  MoveL 7193 to (-68.89, 13.92, -254.44) mm, rotated rx 81.04 ry 30.21 rz 20.91 deg; joints [-4.482, -3.085, 63.14, 103.728, 105.898, 55.876, -153.967]
  MoveL 7194 to (-69.18, 14.22, -254.5) mm, rotated rx 81.04 ry 30.21 rz 20.91 deg; joints [-4.474, -3.068, 63.132, 103.732, 105.896, 55.866, -153.967]
  MoveL 7195 to (-69.51, 14.55, -254.53) mm, rotated rx 81.04 ry 30.21 rz 20.91 deg; joints [-4.464, -3.052, 63.128, 103.737, 105.894, 55.854, -153.967]
  MoveL 7196 to (-69.85, 14.88, -254.55) mm, rotated rx 81.04 ry 30.21 rz 20.91 deg; joints [-4.454, -3.036, 63.123, 103.743, 105.892, 55.84, -153.967]
  MoveL 7197 to (-70.15, 15.2, -254.6) mm, rotated rx 81.04 ry 30.21 rz 20.91 deg; joints [-4.445, -3.02, 63.118, 103.747, 105.89, 55.829, -153.967]
  MoveL 7198 to (-70.42, 15.5, -254.66) mm, rotated rx 81.04 ry 30.21 rz 20.91 deg; joints [-4.438, -3.004, 63.111, 103.751, 105.889, 55.819, -153.967]
  MoveL 7199 to (-70.7, 15.8, -254.71) mm, rotated rx 81.04 ry 30.21 rz 20.91 deg; joints [-4.43, -2.989, 63.105, 103.755, 105.887, 55.808, -153.967]
  MoveL 7200 to (-71.01, 16.11, -254.74) mm, rotated rx 81.04 ry 30.21 rz 20.91 deg; joints [-4.421, -2.973, 63.1, 103.759, 105.885, 55.796, -153.967]
  MoveL 7201 to (-71.4, 16.46, -254.74) mm, rotated rx 81.04 ry 30.21 rz 20.91 deg; joints [-4.409, -2.958, 63.098, 103.766, 105.882, 55.781, -153.967]
  MoveL 7202 to (-73.37, 18.61, -255.1) mm, rotated rx 81.04 ry 30.21 rz 20.91 deg; joints [-4.352, -2.846, 63.055, 103.794, 105.871, 55.705, -153.967]
  MoveL 7203 to (-74.08, 19.69, -255.54) mm, rotated rx 81.04 ry 30.21 rz 20.91 deg; joints [-4.336, -2.778, 63.012, 103.801, 105.869, 55.678, -153.967]
  MoveL 7204 to (-74.6, 20.77, -256.16) mm, rotated rx 81.04 ry 30.21 rz 20.91 deg; joints [-4.327, -2.701, 62.953, 103.803, 105.87, 55.658, -153.967]
  MoveL 7205 to (-75.09, 22.93, -257.95) mm, rotated rx 81.04 ry 30.21 rz 20.91 deg; joints [-4.333, -2.52, 62.791, 103.793, 105.877, 55.64, -153.967]
  MoveL 7206 to (-74.84, 25.11, -260.44) mm, rotated rx 81.04 ry 30.21 rz 20.91 deg; joints [-4.37, -2.305, 62.568, 103.764, 105.893, 55.652, -153.967]
  MoveL 7207 to (-74.04, 26.72, -262.93) mm, rotated rx 81.04 ry 30.21 rz 20.91 deg; joints [-4.424, -2.113, 62.345, 103.728, 105.912, 55.691, -153.967]
  MoveL 7208 to (-73.5, 27.09, -263.91) mm, rotated rx 81.04 ry 30.21 rz 20.91 deg; joints [-4.452, -2.047, 62.256, 103.711, 105.92, 55.717, -153.967]
  MoveL 7209 to (-72.87, 27.18, -264.71) mm, rotated rx 81.04 ry 30.21 rz 20.91 deg; joints [-4.481, -2.001, 62.182, 103.694, 105.927, 55.749, -153.967]
  MoveL 7210 to (-72.52, 27.12, -265.05) mm, rotated rx 81.04 ry 30.21 rz 20.91 deg; joints [-4.496, -1.986, 62.151, 103.687, 105.93, 55.767, -153.967]
  MoveL 7211 to (-72.14, 26.98, -265.34) mm, rotated rx 81.04 ry 30.21 rz 20.91 deg; joints [-4.51, -1.976, 62.123, 103.679, 105.933, 55.786, -153.967]
  MoveL 7212 to (-71.33, 26.5, -265.78) mm, rotated rx 81.04 ry 30.21 rz 20.91 deg; joints [-4.541, -1.97, 62.08, 103.664, 105.939, 55.828, -153.967]
  MoveL 7213 to (-70.42, 25.73, -266.05) mm, rotated rx 81.04 ry 30.21 rz 20.91 deg; joints [-4.572, -1.985, 62.052, 103.65, 105.944, 55.876, -153.967]
  MoveL 7214 to (-69.43, 24.68, -266.14) mm, rotated rx 81.04 ry 30.21 rz 20.91 deg; joints [-4.603, -2.02, 62.039, 103.637, 105.948, 55.928, -153.967]
  MoveL 7215 to (-67.7, 22.71, -266.14) mm, rotated rx 81.04 ry 30.21 rz 20.91 deg; joints [-4.656, -2.094, 62.03, 103.617, 105.954, 56.018, -153.967]
  MoveL 7216 to (-67.43, 22.36, -266.11) mm, rotated rx 81.04 ry 30.21 rz 20.91 deg; joints [-4.664, -2.109, 62.032, 103.614, 105.955, 56.032, -153.967]
  MoveL 7217 to (-67.18, 22.04, -266.06) mm, rotated rx 81.04 ry 30.21 rz 20.91 deg; joints [-4.671, -2.124, 62.035, 103.611, 105.956, 56.045, -153.967]
  MoveL 7218 to (-66.95, 21.73, -265.99) mm, rotated rx 81.04 ry 30.21 rz 20.91 deg; joints [-4.677, -2.14, 62.041, 103.609, 105.956, 56.056, -153.967]
  MoveL 7219 to (-66.69, 21.39, -265.94) mm, rotated rx 81.04 ry 30.21 rz 20.91 deg; joints [-4.685, -2.155, 62.044, 103.606, 105.957, 56.069, -153.967]
  MoveL 7220 to (-66.38, 21, -265.9) mm, rotated rx 81.04 ry 30.21 rz 20.91 deg; joints [-4.694, -2.172, 62.046, 103.602, 105.958, 56.085, -153.967]
  MoveL 7221 to (-66.06, 20.59, -265.84) mm, rotated rx 81.04 ry 30.21 rz 20.91 deg; joints [-4.703, -2.191, 62.05, 103.599, 105.959, 56.102, -153.967]
  MoveL 7222 to (-65.71, 20.17, -265.83) mm, rotated rx 81.04 ry 30.21 rz 20.91 deg; joints [-4.713, -2.208, 62.05, 103.595, 105.96, 56.12, -153.967]
  MoveL 7223 to (-65.28, 19.69, -265.84) mm, rotated rx 81.04 ry 30.21 rz 20.91 deg; joints [-4.727, -2.225, 62.046, 103.59, 105.961, 56.143, -153.967]
  MoveL 7224 to (-64.69, 19.05, -265.91) mm, rotated rx 81.04 ry 30.21 rz 20.91 deg; joints [-4.745, -2.244, 62.035, 103.583, 105.963, 56.176, -153.967]
  MoveL 7225 to (-64.35, 18.66, -265.91) mm, rotated rx 81.04 ry 30.21 rz 20.91 deg; joints [-4.756, -2.259, 62.033, 103.579, 105.965, 56.194, -153.967]
  MoveL 7226 to (-64.02, 18.28, -265.9) mm, rotated rx 81.04 ry 30.21 rz 20.91 deg; joints [-4.766, -2.273, 62.031, 103.575, 105.966, 56.211, -153.967]
  MoveL 7227 to (-63.72, 17.92, -265.88) mm, rotated rx 81.04 ry 30.21 rz 20.91 deg; joints [-4.775, -2.288, 62.032, 103.571, 105.967, 56.227, -153.967]
  MoveL 7228 to (-63.47, 17.59, -265.83) mm, rotated rx 81.04 ry 30.21 rz 20.91 deg; joints [-4.782, -2.303, 62.035, 103.569, 105.967, 56.24, -153.967]
  MoveL 7229 to (-63.25, 17.26, -265.77) mm, rotated rx 81.04 ry 30.21 rz 20.91 deg; joints [-4.788, -2.318, 62.038, 103.567, 105.968, 56.252, -153.967]
  MoveL 7230 to (-63.04, 16.89, -265.72) mm, rotated rx 81.04 ry 30.21 rz 20.91 deg; joints [-4.794, -2.332, 62.037, 103.566, 105.967, 56.269, -153.967]
  MoveL 7231 to (-62.88, 16.51, -265.66) mm, rotated rx 81.04 ry 30.21 rz 20.91 deg; joints [-4.798, -2.346, 62.034, 103.568, 105.965, 56.286, -153.967]
  MoveL 7232 to (-62.86, 16.29, -265.5) mm, rotated rx 81.04 ry 30.21 rz 20.91 deg; joints [-4.797, -2.362, 62.047, 103.57, 105.964, 56.289, -153.967]
  MoveL 7233 to (-62.95, 16.34, -265.19) mm, rotated rx 81.04 ry 30.21 rz 20.91 deg; joints [-4.79, -2.384, 62.088, 103.57, 105.965, 56.269, -153.967]
  MoveL 7234 to (-63.19, 16.71, -264.7) mm, rotated rx 81.04 ry 30.21 rz 20.91 deg; joints [-4.777, -2.412, 62.163, 103.567, 105.97, 56.22, -153.967]
  MoveL 7235 to (-63.04, 15.84, -263.84) mm, rotated rx 81.04 ry 30.21 rz 20.91 deg; joints [-4.772, -2.493, 62.244, 103.572, 105.967, 56.22, -153.967]
  MoveL 7236 to (-62.5, 11.6, -263.84) mm, rotated rx 81.04 ry 30.21 rz 20.91 deg; joints [-4.787, -2.557, 62.06, 103.628, 105.916, 56.472, -153.967]
  MoveL 7237 to (-62.26, 9.62, -263.78) mm, rotated rx 81.04 ry 30.21 rz 20.91 deg; joints [-4.793, -2.592, 61.982, 103.654, 105.893, 56.586, -153.967]
  MoveL 7238 to (-62.02, 7.64, -263.63) mm, rotated rx 81.04 ry 30.21 rz 20.91 deg; joints [-4.798, -2.632, 61.914, 103.68, 105.87, 56.696, -153.967]
  MoveL 7239 to (-61.76, 5.36, -263.43) mm, rotated rx 81.04 ry 30.21 rz 20.91 deg; joints [-4.803, -2.68, 61.84, 103.709, 105.843, 56.821, -153.967]
  MoveL 7240 to (-61.5, 3.21, -263.22) mm, rotated rx 81.04 ry 30.21 rz 20.91 deg; joints [-4.808, -2.727, 61.772, 103.737, 105.818, 56.937, -153.967]
  MoveL 7241 to (-61.23, 1.04, -263.12) mm, rotated rx 81.04 ry 30.21 rz 20.91 deg; joints [-4.814, -2.766, 61.689, 103.766, 105.792, 57.061, -153.967]
  MoveL 7242 to (-60.96, -1.08, -263.12) mm, rotated rx 81.04 ry 30.21 rz 20.91 deg; joints [-4.822, -2.796, 61.593, 103.794, 105.766, 57.189, -153.967]
  MoveL 7243 to (-60.71, -3.05, -263.05) mm, rotated rx 81.04 ry 30.21 rz 20.91 deg; joints [-4.828, -2.828, 61.513, 103.82, 105.743, 57.303, -153.967]
  MoveL 7244 to (-60.47, -4.91, -262.94) mm, rotated rx 81.04 ry 30.21 rz 20.91 deg; joints [-4.834, -2.863, 61.444, 103.843, 105.721, 57.408, -153.967]
  MoveL 7245 to (-60.21, -6.93, -262.87) mm, rotated rx 81.04 ry 30.21 rz 20.91 deg; joints [-4.84, -2.896, 61.361, 103.87, 105.696, 57.527, -153.967]
  MoveL 7246 to (-59.94, -9.05, -262.69) mm, rotated rx 81.04 ry 30.21 rz 20.91 deg; joints [-4.846, -2.939, 61.288, 103.897, 105.671, 57.644, -153.967]
  MoveL 7247 to (-59.39, -13.28, -262.51) mm, rotated rx 81.04 ry 30.21 rz 20.91 deg; joints [-4.859, -3.01, 61.117, 103.952, 105.62, 57.89, -153.967]
  MoveL 7248 to (-59.11, -15.4, -262.33) mm, rotated rx 81.04 ry 30.21 rz 20.91 deg; joints [-4.864, -3.052, 61.043, 103.979, 105.595, 58.007, -153.967]
  MoveL 7249 to (-58.82, -17.51, -262.15) mm, rotated rx 81.04 ry 30.21 rz 20.91 deg; joints [-4.87, -3.094, 60.969, 104.005, 105.57, 58.125, -153.967]
  MoveL 7250 to (-58.55, -19.63, -262.15) mm, rotated rx 81.04 ry 30.21 rz 20.91 deg; joints [-4.878, -3.12, 60.868, 104.034, 105.543, 58.254, -153.967]
  MoveL 7251 to (-58.26, -21.75, -261.97) mm, rotated rx 81.04 ry 30.21 rz 20.91 deg; joints [-4.884, -3.162, 60.793, 104.06, 105.517, 58.372, -153.967]
  MoveL 7252 to (-57.97, -23.86, -261.79) mm, rotated rx 81.04 ry 30.21 rz 20.91 deg; joints [-4.89, -3.203, 60.717, 104.086, 105.492, 58.491, -153.967]
  MoveL 7253 to (-57.7, -25.98, -261.79) mm, rotated rx 81.04 ry 30.21 rz 20.91 deg; joints [-4.898, -3.228, 60.615, 104.115, 105.465, 58.62, -153.967]
  MoveL 7254 to (-57.38, -27.9, -261.6) mm, rotated rx 81.04 ry 30.21 rz 20.91 deg; joints [-4.904, -3.269, 60.553, 104.137, 105.443, 58.725, -153.967]
  MoveL 7255 to (-57.03, -29.57, -261.28) mm, rotated rx 81.04 ry 30.21 rz 20.91 deg; joints [-4.911, -3.319, 60.523, 104.153, 105.427, 58.807, -153.967]
  MoveL 7256 to (-56.65, -31.05, -260.81) mm, rotated rx 81.04 ry 30.21 rz 20.91 deg; joints [-4.917, -3.381, 60.526, 104.164, 105.416, 58.866, -153.967]
  MoveL 7257 to (-56.59, -30.11, -260.05) mm, rotated rx 81.04 ry 30.21 rz 20.91 deg; joints [-4.91, -3.437, 60.688, 104.141, 105.439, 58.758, -153.967]
  MoveL 7258 to (-56.59, -30.52, -260.04) mm, rotated rx 81.04 ry 30.21 rz 20.91 deg; joints [-4.91, -3.441, 60.667, 104.148, 105.432, 58.784, -153.967]
  MoveC 7259 to (-57.91, -33.82, -260.04) mm, rotated rx 81.04 ry 30.21 rz 20.91 deg; joints [-4.868, -3.427, 60.415, 104.245, 105.352, 59.017, -153.967] to (-59.51, -36.99, -260.04) mm, rotated rx 81.04 ry 30.21 rz 20.91 deg; joints [-4.819, -3.402, 60.155, 104.347, 105.268, 59.247, -153.967]
  MoveL 7260 to (-59.51, -36.99, -260.04) mm, rotated rx 81.04 ry 30.21 rz 20.91 deg; joints [-4.819, -3.402, 60.155, 104.347, 105.268, 59.247, -153.967]
  MoveL 7261 to (-59.71, -37.42, -260.02) mm, rotated rx 81.04 ry 30.21 rz 20.91 deg; joints [-4.812, -3.401, 60.123, 104.36, 105.257, 59.276, -153.967]
  MoveL 7262 to (-59.88, -37.81, -259.97) mm, rotated rx 81.04 ry 30.21 rz 20.91 deg; joints [-4.807, -3.403, 60.1, 104.371, 105.247, 59.301, -153.967]
  MoveL 7263 to (-60.03, -38.19, -259.91) mm, rotated rx 81.04 ry 30.21 rz 20.91 deg; joints [-4.801, -3.406, 60.08, 104.382, 105.239, 59.324, -153.967]
  MoveL 7264 to (-60.2, -38.59, -259.86) mm, rotated rx 81.04 ry 30.21 rz 20.91 deg; joints [-4.795, -3.407, 60.054, 104.394, 105.229, 59.35, -153.967]
  MoveL 7265 to (-60.4, -39.02, -259.83) mm, rotated rx 81.04 ry 30.21 rz 20.91 deg; joints [-4.789, -3.407, 60.024, 104.407, 105.218, 59.379, -153.967]
  MoveL 7266 to (-60.62, -39.49, -259.82) mm, rotated rx 81.04 ry 30.21 rz 20.91 deg; joints [-4.782, -3.405, 59.988, 104.421, 105.206, 59.412, -153.967]
  MoveL 7267 to (-61.09, -40.42, -259.82) mm, rotated rx 81.04 ry 30.21 rz 20.91 deg; joints [-4.767, -3.397, 59.91, 104.451, 105.181, 59.48, -153.967]
  MoveL 7268 to (-61.79, -41.7, -259.91) mm, rotated rx 81.04 ry 30.21 rz 20.91 deg; joints [-4.746, -3.377, 59.788, 104.495, 105.144, 59.579, -153.967]
  MoveL 7269 to (-62.48, -42.68, -260.18) mm, rotated rx 81.04 ry 30.21 rz 20.91 deg; joints [-4.728, -3.339, 59.656, 104.534, 105.111, 59.671, -153.967]
  MoveL 7270 to (-63.15, -43.38, -260.64) mm, rotated rx 81.04 ry 30.21 rz 20.91 deg; joints [-4.713, -3.286, 59.516, 104.568, 105.081, 59.756, -153.967]
  MoveL 7271 to (-63.8, -43.79, -261.28) mm, rotated rx 81.04 ry 30.21 rz 20.91 deg; joints [-4.7, -3.215, 59.367, 104.599, 105.054, 59.833, -153.967]
  MoveL 7272 to (-64.44, -43.91, -262.1) mm, rotated rx 81.04 ry 30.21 rz 20.91 deg; joints [-4.69, -3.128, 59.208, 104.626, 105.031, 59.903, -153.967]
  MoveL 7273 to (-65.06, -43.75, -263.11) mm, rotated rx 81.04 ry 30.21 rz 20.91 deg; joints [-4.683, -3.024, 59.041, 104.648, 105.01, 59.965, -153.967]
  MoveL 7274 to (-66.25, -42.54, -265.67) mm, rotated rx 81.04 ry 30.21 rz 20.91 deg; joints [-4.676, -2.765, 58.677, 104.681, 104.98, 60.069, -153.967]
  MoveL 7275 to (-67.04, -40.65, -268.23) mm, rotated rx 81.04 ry 30.21 rz 20.91 deg; joints [-4.681, -2.513, 58.372, 104.69, 104.969, 60.123, -153.967]
  MoveL 7276 to (-67.17, -39.63, -269.23) mm, rotated rx 81.04 ry 30.21 rz 20.91 deg; joints [-4.688, -2.418, 58.278, 104.684, 104.974, 60.123, -153.967]
  MoveL 7277 to (-67.12, -38.54, -270.06) mm, rotated rx 81.04 ry 30.21 rz 20.91 deg; joints [-4.699, -2.343, 58.224, 104.67, 104.985, 60.104, -153.967]
  MoveL 7278 to (-66.89, -37.4, -270.7) mm, rotated rx 81.04 ry 30.21 rz 20.91 deg; joints [-4.714, -2.289, 58.209, 104.649, 105.003, 60.068, -153.967]
  MoveL 7279 to (-66.48, -36.21, -271.15) mm, rotated rx 81.04 ry 30.21 rz 20.91 deg; joints [-4.732, -2.256, 58.233, 104.619, 105.027, 60.012, -153.967]
  MoveL 7280 to (-65.12, -33.65, -271.52) mm, rotated rx 81.04 ry 30.21 rz 20.91 deg; joints [-4.778, -2.251, 58.4, 104.538, 105.095, 59.847, -153.967]
  MoveL 7281 to (-64.55, -32.77, -271.52) mm, rotated rx 81.04 ry 30.21 rz 20.91 deg; joints [-4.795, -2.263, 58.481, 104.506, 105.122, 59.78, -153.967]
  MoveL 7282 to (-64.27, -32.32, -271.53) mm, rotated rx 81.04 ry 30.21 rz 20.91 deg; joints [-4.804, -2.268, 58.521, 104.49, 105.135, 59.747, -153.967]
  MoveL 7283 to (-64.03, -31.92, -271.55) mm, rotated rx 81.04 ry 30.21 rz 20.91 deg; joints [-4.812, -2.272, 58.554, 104.476, 105.147, 59.718, -153.967]
  MoveL 7284 to (-63.82, -31.55, -271.6) mm, rotated rx 81.04 ry 30.21 rz 20.91 deg; joints [-4.819, -2.271, 58.579, 104.464, 105.157, 59.694, -153.967]
  MoveL 7285 to (-63.63, -31.19, -271.65) mm, rotated rx 81.04 ry 30.21 rz 20.91 deg; joints [-4.825, -2.27, 58.601, 104.453, 105.166, 59.671, -153.967]
  MoveL 7286 to (-63.43, -30.83, -271.7) mm, rotated rx 81.04 ry 30.21 rz 20.91 deg; joints [-4.832, -2.27, 58.626, 104.441, 105.176, 59.647, -153.967]
  MoveL 7287 to (-63.18, -30.43, -271.72) mm, rotated rx 81.04 ry 30.21 rz 20.91 deg; joints [-4.84, -2.273, 58.659, 104.427, 105.188, 59.618, -153.967]
  MoveL 7288 to (-62.91, -30.01, -271.73) mm, rotated rx 81.04 ry 30.21 rz 20.91 deg; joints [-4.848, -2.278, 58.696, 104.412, 105.2, 59.587, -153.967]
  MoveL 7289 to (-62.61, -29.54, -271.72) mm, rotated rx 81.04 ry 30.21 rz 20.91 deg; joints [-4.858, -2.285, 58.739, 104.395, 105.214, 59.551, -153.967]
  MoveL 7290 to (-62.33, -29.09, -271.73) mm, rotated rx 81.04 ry 30.21 rz 20.91 deg; joints [-4.866, -2.29, 58.778, 104.379, 105.228, 59.518, -153.967]
  MoveL 7291 to (-62.07, -28.67, -271.75) mm, rotated rx 81.04 ry 30.21 rz 20.91 deg; joints [-4.875, -2.293, 58.813, 104.364, 105.24, 59.488, -153.967]
  MoveL 7292 to (-61.83, -28.26, -271.8) mm, rotated rx 81.04 ry 30.21 rz 20.91 deg; joints [-4.883, -2.293, 58.842, 104.35, 105.251, 59.461, -153.967]
  MoveL 7293 to (-61.59, -27.82, -271.88) mm, rotated rx 81.04 ry 30.21 rz 20.91 deg; joints [-4.891, -2.291, 58.868, 104.336, 105.263, 59.433, -153.967]
  MoveL 7294 to (-61.29, -27.29, -271.94) mm, rotated rx 81.04 ry 30.21 rz 20.91 deg; joints [-4.901, -2.291, 58.905, 104.318, 105.277, 59.398, -153.967]
  MoveL 7295 to (-61, -26.81, -271.96) mm, rotated rx 81.04 ry 30.21 rz 20.91 deg; joints [-4.91, -2.295, 58.945, 104.301, 105.291, 59.363, -153.967]
  MoveL 7296 to (-60.71, -26.36, -271.96) mm, rotated rx 81.04 ry 30.21 rz 20.91 deg; joints [-4.919, -2.301, 58.985, 104.285, 105.304, 59.33, -153.967]
  MoveL 7297 to (-60.43, -25.92, -271.96) mm, rotated rx 81.04 ry 30.21 rz 20.91 deg; joints [-4.928, -2.306, 59.025, 104.269, 105.317, 59.296, -153.967]
  MoveL 7298 to (-60.09, -25.36, -271.97) mm, rotated rx 81.04 ry 30.21 rz 20.91 deg; joints [-4.939, -2.311, 59.073, 104.249, 105.333, 59.255, -153.967]
  MoveL 7299 to (-59.8, -24.85, -271.98) mm, rotated rx 81.04 ry 30.21 rz 20.91 deg; joints [-4.948, -2.316, 59.115, 104.232, 105.348, 59.218, -153.967]
  MoveL 7300 to (-59.58, -24.39, -271.99) mm, rotated rx 81.04 ry 30.21 rz 20.91 deg; joints [-4.955, -2.318, 59.151, 104.217, 105.359, 59.186, -153.967]
  MoveL 7301 to (-59.48, -24.06, -271.99) mm, rotated rx 81.04 ry 30.21 rz 20.91 deg; joints [-4.958, -2.319, 59.174, 104.209, 105.367, 59.163, -153.967]
  MoveL 7302 to (-59.44, -23.8, -271.99) mm, rotated rx 81.04 ry 30.21 rz 20.91 deg; joints [-4.959, -2.318, 59.191, 104.203, 105.372, 59.145, -153.967]
  MoveL 7303 to (-59.56, -24.73, -272.58) mm, rotated rx 81.04 ry 30.21 rz 20.91 deg; joints [-4.962, -2.272, 59.047, 104.227, 105.349, 59.244, -153.967]
  MoveL 7304 to (-59.85, -23.43, -273.11) mm, rotated rx 81.04 ry 30.21 rz 20.91 deg; joints [-4.959, -2.209, 59.028, 104.217, 105.358, 59.2, -153.967]
  MoveL 7305 to (-60.06, -21.88, -273.49) mm, rotated rx 81.04 ry 30.21 rz 20.91 deg; joints [-4.958, -2.159, 59.048, 104.2, 105.375, 59.129, -153.967]
  MoveL 7306 to (-60.2, -20.04, -273.75) mm, rotated rx 81.04 ry 30.21 rz 20.91 deg; joints [-4.957, -2.119, 59.106, 104.174, 105.399, 59.031, -153.967]
  MoveL 7307 to (-60.27, -17.98, -273.88) mm, rotated rx 81.04 ry 30.21 rz 20.91 deg; joints [-4.957, -2.091, 59.199, 104.141, 105.428, 58.909, -153.967]
  MoveL 7308 to (-60.32, -15.88, -273.97) mm, rotated rx 81.04 ry 30.21 rz 20.91 deg; joints [-4.958, -2.065, 59.298, 104.107, 105.459, 58.782, -153.967]
  MoveL 7309 to (-60.42, -11.62, -274.15) mm, rotated rx 81.04 ry 30.21 rz 20.91 deg; joints [-4.958, -2.011, 59.501, 104.038, 105.522, 58.525, -153.967]
  MoveL 7310 to (-60.47, -9.48, -274.33) mm, rotated rx 81.04 ry 30.21 rz 20.91 deg; joints [-4.96, -1.977, 59.588, 104.004, 105.552, 58.403, -153.967]
  MoveL 7311 to (-60.56, -5.22, -274.51) mm, rotated rx 81.04 ry 30.21 rz 20.91 deg; joints [-4.961, -1.921, 59.787, 103.935, 105.614, 58.147, -153.967]
  MoveL 7312 to (-60.6, -3.08, -274.69) mm, rotated rx 81.04 ry 30.21 rz 20.91 deg; joints [-4.962, -1.886, 59.872, 103.9, 105.644, 58.025, -153.967]
  MoveL 7313 to (-60.64, -0.95, -274.78) mm, rotated rx 81.04 ry 30.21 rz 20.91 deg; joints [-4.963, -1.857, 59.97, 103.866, 105.674, 57.898, -153.967]
  MoveL 7314 to (-60.66, 1.02, -274.99) mm, rotated rx 81.04 ry 30.21 rz 20.91 deg; joints [-4.966, -1.821, 60.044, 103.833, 105.702, 57.787, -153.967]
  MoveL 7315 to (-60.7, 3.38, -275.14) mm, rotated rx 81.04 ry 30.21 rz 20.91 deg; joints [-4.967, -1.785, 60.144, 103.795, 105.735, 57.65, -153.967]
  MoveL 7316 to (-60.75, 5.94, -275.26) mm, rotated rx 81.04 ry 30.21 rz 20.91 deg; joints [-4.968, -1.748, 60.258, 103.753, 105.772, 57.498, -153.967]
  MoveL 7317 to (-60.79, 8.08, -275.26) mm, rotated rx 81.04 ry 30.21 rz 20.91 deg; joints [-4.968, -1.726, 60.367, 103.717, 105.803, 57.366, -153.967]
  MoveL 7318 to (-60.82, 10.11, -275.33) mm, rotated rx 81.04 ry 30.21 rz 20.91 deg; joints [-4.968, -1.698, 60.459, 103.684, 105.831, 57.244, -153.967]
  MoveL 7319 to (-60.83, 11.94, -275.51) mm, rotated rx 81.04 ry 30.21 rz 20.91 deg; joints [-4.971, -1.665, 60.528, 103.653, 105.857, 57.142, -153.967]
  MoveL 7320 to (-60.82, 13.81, -275.72) mm, rotated rx 81.04 ry 30.21 rz 20.91 deg; joints [-4.974, -1.628, 60.594, 103.622, 105.883, 57.039, -153.967]
  MoveL 7321 to (-60.85, 16.17, -275.85) mm, rotated rx 81.04 ry 30.21 rz 20.91 deg; joints [-4.976, -1.591, 60.692, 103.584, 105.915, 56.902, -153.967]
  MoveL 7322 to (-60.89, 18.75, -275.96) mm, rotated rx 81.04 ry 30.21 rz 20.91 deg; joints [-4.977, -1.553, 60.805, 103.541, 105.951, 56.75, -153.967]
  MoveL 7323 to (-60.97, 23.02, -275.96) mm, rotated rx 81.04 ry 30.21 rz 20.91 deg; joints [-4.976, -1.504, 61.014, 103.469, 106.011, 56.488, -153.967]
  MoveL 7324 to (-60.73, 23.23, -276.66) mm, rotated rx 81.04 ry 30.21 rz 20.91 deg; joints [-4.991, -1.452, 60.938, 103.463, 106.013, 56.514, -153.967]
  MoveL 7325 to (-60.61, 22.95, -277) mm, rotated rx 81.04 ry 30.21 rz 20.91 deg; joints [-4.999, -1.431, 60.882, 103.467, 106.009, 56.551, -153.967]
  MoveL 7326 to (-60.59, 22.94, -277.22) mm, rotated rx 81.04 ry 30.21 rz 20.91 deg; joints [-5.002, -1.414, 60.852, 103.468, 106.007, 56.565, -153.967]
  MoveL 7327 to (-60.68, 23.19, -277.33) mm, rotated rx 81.04 ry 30.21 rz 20.91 deg; joints [-5.001, -1.399, 60.844, 103.468, 106.008, 56.558, -153.967]
  MoveL 7328 to (-60.89, 23.59, -277.36) mm, rotated rx 81.04 ry 30.21 rz 20.91 deg; joints [-4.995, -1.386, 60.848, 103.467, 106.009, 56.539, -153.967]
  MoveL 7329 to (-61.13, 24.01, -277.39) mm, rotated rx 81.04 ry 30.21 rz 20.91 deg; joints [-4.988, -1.372, 60.853, 103.468, 106.01, 56.519, -153.967]
  MoveL 7330 to (-61.36, 24.37, -277.43) mm, rotated rx 81.04 ry 30.21 rz 20.91 deg; joints [-4.981, -1.358, 60.853, 103.469, 106.01, 56.504, -153.967]
  MoveL 7331 to (-61.56, 24.72, -277.5) mm, rotated rx 81.04 ry 30.21 rz 20.91 deg; joints [-4.976, -1.342, 60.85, 103.47, 106.011, 56.49, -153.967]
  MoveL 7332 to (-61.77, 25.07, -277.56) mm, rotated rx 81.04 ry 30.21 rz 20.91 deg; joints [-4.97, -1.327, 60.848, 103.471, 106.011, 56.476, -153.967]
  MoveL 7333 to (-62.01, 25.45, -277.6) mm, rotated rx 81.04 ry 30.21 rz 20.91 deg; joints [-4.964, -1.313, 60.849, 103.472, 106.011, 56.46, -153.967]
  MoveL 7334 to (-62.3, 25.88, -277.62) mm, rotated rx 81.04 ry 30.21 rz 20.91 deg; joints [-4.955, -1.297, 60.853, 103.474, 106.011, 56.439, -153.967]
  MoveL 7335 to (-62.57, 26.34, -277.69) mm, rotated rx 81.04 ry 30.21 rz 20.91 deg; joints [-4.947, -1.279, 60.852, 103.476, 106.012, 56.421, -153.967]
  MoveL 7336 to (-62.86, 26.77, -277.72) mm, rotated rx 81.04 ry 30.21 rz 20.91 deg; joints [-4.939, -1.262, 60.854, 103.477, 106.012, 56.401, -153.967]
  MoveL 7337 to (-63.15, 27.2, -277.72) mm, rotated rx 81.04 ry 30.21 rz 20.91 deg; joints [-4.93, -1.248, 60.859, 103.479, 106.012, 56.38, -153.967]
  MoveL 7338 to (-63.45, 27.63, -277.72) mm, rotated rx 81.04 ry 30.21 rz 20.91 deg; joints [-4.921, -1.235, 60.865, 103.481, 106.012, 56.359, -153.967]
  MoveL 7339 to (-63.86, 28.19, -277.69) mm, rotated rx 81.04 ry 30.21 rz 20.91 deg; joints [-4.908, -1.219, 60.877, 103.484, 106.012, 56.33, -153.967]
  MoveL 7340 to (-64.25, 28.72, -277.66) mm, rotated rx 81.04 ry 30.21 rz 20.91 deg; joints [-4.896, -1.203, 60.887, 103.487, 106.012, 56.303, -153.967]
  MoveL 7341 to (-64.6, 29.21, -277.65) mm, rotated rx 81.04 ry 30.21 rz 20.91 deg; joints [-4.886, -1.188, 60.894, 103.49, 106.012, 56.278, -153.967]
  MoveL 7342 to (-64.85, 29.61, -277.69) mm, rotated rx 81.04 ry 30.21 rz 20.91 deg; joints [-4.878, -1.173, 60.895, 103.491, 106.013, 56.261, -153.967]
  MoveL 7343 to (-65.06, 29.96, -277.75) mm, rotated rx 81.04 ry 30.21 rz 20.91 deg; joints [-4.873, -1.157, 60.893, 103.492, 106.013, 56.247, -153.967]
  MoveL 7344 to (-65.27, 30.31, -277.81) mm, rotated rx 81.04 ry 30.21 rz 20.91 deg; joints [-4.867, -1.143, 60.892, 103.493, 106.013, 56.232, -153.967]
  MoveL 7345 to (-65.51, 30.69, -277.84) mm, rotated rx 81.04 ry 30.21 rz 20.91 deg; joints [-4.86, -1.128, 60.893, 103.495, 106.014, 56.216, -153.967]
  MoveL 7346 to (-66.41, 31.98, -277.84) mm, rotated rx 81.04 ry 30.21 rz 20.91 deg; joints [-4.833, -1.086, 60.91, 103.501, 106.014, 56.153, -153.967]
  MoveL 7347 to (-67.87, 34.47, -278.22) mm, rotated rx 81.04 ry 30.21 rz 20.91 deg; joints [-4.793, -0.983, 60.902, 103.507, 106.017, 56.051, -153.967]
  MoveL 7348 to (-68.33, 35.63, -278.69) mm, rotated rx 81.04 ry 30.21 rz 20.91 deg; joints [-4.784, -0.917, 60.868, 103.506, 106.02, 56.019, -153.967]
  MoveL 7349 to (-68.62, 36.74, -279.35) mm, rotated rx 81.04 ry 30.21 rz 20.91 deg; joints [-4.783, -0.842, 60.813, 103.501, 106.024, 55.998, -153.967]
  MoveL 7350 to (-68.73, 37.79, -280.19) mm, rotated rx 81.04 ry 30.21 rz 20.91 deg; joints [-4.79, -0.757, 60.738, 103.493, 106.03, 55.99, -153.967]
  MoveL 7351 to (-68.66, 38.79, -281.23) mm, rotated rx 81.04 ry 30.21 rz 20.91 deg; joints [-4.804, -0.664, 60.642, 103.481, 106.036, 55.993, -153.967]
  MoveL 7352 to (-67.99, 40.62, -283.87) mm, rotated rx 81.04 ry 30.21 rz 20.91 deg; joints [-4.856, -0.448, 60.387, 103.449, 106.052, 56.038, -153.967]
  MoveL 7353 to (-66.9, 41.78, -286.5) mm, rotated rx 81.04 ry 30.21 rz 20.91 deg; joints [-4.92, -0.251, 60.121, 103.416, 106.067, 56.118, -153.967]
  MoveL 7354 to (-66.31, 41.93, -287.54) mm, rotated rx 81.04 ry 30.21 rz 20.91 deg; joints [-4.95, -0.183, 60.01, 103.403, 106.072, 56.164, -153.967]
  MoveL 7355 to (-65.68, 41.81, -288.39) mm, rotated rx 81.04 ry 30.21 rz 20.91 deg; joints [-4.979, -0.134, 59.914, 103.392, 106.075, 56.215, -153.967]
  MoveL 7356 to (-65.02, 41.41, -289.05) mm, rotated rx 81.04 ry 30.21 rz 20.91 deg; joints [-5.006, -0.104, 59.833, 103.383, 106.077, 56.271, -153.967]
  MoveL 7357 to (-64.33, 40.72, -289.52) mm, rotated rx 81.04 ry 30.21 rz 20.91 deg; joints [-5.033, -0.094, 59.767, 103.377, 106.077, 56.33, -153.967]
  MoveL 7358 to (-63.61, 39.75, -289.8) mm, rotated rx 81.04 ry 30.21 rz 20.91 deg; joints [-5.058, -0.104, 59.717, 103.373, 106.075, 56.394, -153.967]
  MoveL 7359 to (-62.85, 38.51, -289.89) mm, rotated rx 81.04 ry 30.21 rz 20.91 deg; joints [-5.082, -0.134, 59.682, 103.371, 106.072, 56.463, -153.967]
  MoveL 7360 to (-62.6, 38.05, -289.89) mm, rotated rx 81.04 ry 30.21 rz 20.91 deg; joints [-5.089, -0.147, 59.672, 103.371, 106.071, 56.486, -153.967]
  MoveL 7361 to (-62.38, 37.64, -289.87) mm, rotated rx 81.04 ry 30.21 rz 20.91 deg; joints [-5.096, -0.16, 59.666, 103.371, 106.069, 56.506, -153.967]
  MoveL 7362 to (-62.21, 37.27, -289.83) mm, rotated rx 81.04 ry 30.21 rz 20.91 deg; joints [-5.1, -0.173, 59.665, 103.372, 106.068, 56.522, -153.967]
  MoveL 7363 to (-62.05, 36.91, -289.77) mm, rotated rx 81.04 ry 30.21 rz 20.91 deg; joints [-5.105, -0.187, 59.664, 103.372, 106.067, 56.537, -153.967]
  MoveL 7364 to (-61.86, 36.53, -289.73) mm, rotated rx 81.04 ry 30.21 rz 20.91 deg; joints [-5.11, -0.2, 59.661, 103.373, 106.066, 56.555, -153.967]
  MoveL 7365 to (-61.63, 36.09, -289.7) mm, rotated rx 81.04 ry 30.21 rz 20.91 deg; joints [-5.116, -0.214, 59.655, 103.373, 106.064, 56.576, -153.967]
  MoveL 7366 to (-61.38, 35.63, -289.7) mm, rotated rx 81.04 ry 30.21 rz 20.91 deg; joints [-5.124, -0.227, 59.645, 103.373, 106.063, 56.599, -153.967]
  MoveL 7367 to (-61.16, 35.22, -289.68) mm, rotated rx 81.04 ry 30.21 rz 20.91 deg; joints [-5.13, -0.24, 59.64, 103.373, 106.062, 56.619, -153.967]
  MoveL 7368 to (-60.97, 34.86, -289.63) mm, rotated rx 81.04 ry 30.21 rz 20.91 deg; joints [-5.135, -0.254, 59.639, 103.373, 106.061, 56.634, -153.967]
  MoveL 7369 to (-60.8, 34.51, -289.57) mm, rotated rx 81.04 ry 30.21 rz 20.91 deg; joints [-5.14, -0.268, 59.64, 103.373, 106.06, 56.649, -153.967]
  MoveL 7370 to (-60.61, 34.13, -289.52) mm, rotated rx 81.04 ry 30.21 rz 20.91 deg; joints [-5.145, -0.282, 59.637, 103.373, 106.059, 56.666, -153.967]
  MoveL 7371 to (-60.38, 33.69, -289.5) mm, rotated rx 81.04 ry 30.21 rz 20.91 deg; joints [-5.152, -0.296, 59.632, 103.373, 106.058, 56.686, -153.967]
  MoveL 7372 to (-60.12, 33.24, -289.5) mm, rotated rx 81.04 ry 30.21 rz 20.91 deg; joints [-5.159, -0.309, 59.622, 103.373, 106.056, 56.71, -153.967]
  MoveL 7373 to (-59.71, 32.34, -289.48) mm, rotated rx 81.04 ry 30.21 rz 20.91 deg; joints [-5.171, -0.333, 59.602, 103.375, 106.052, 56.756, -153.967]
  MoveC 7374 to (-59.16, 31.07, -289.48) mm, rotated rx 81.04 ry 30.21 rz 20.91 deg; joints [-5.188, -0.364, 59.567, 103.38, 106.045, 56.824, -153.967] to (-58.47, 29.88, -289.48) mm, rotated rx 81.04 ry 30.21 rz 20.91 deg; joints [-5.208, -0.398, 59.544, 103.379, 106.042, 56.885, -153.967]
  MoveL 7375 to (-58.47, 29.88, -289.47) mm, rotated rx 81.04 ry 30.21 rz 20.91 deg; joints [-5.208, -0.398, 59.546, 103.379, 106.042, 56.884, -153.967]
  MoveL 7376 to (-58.18, 29.28, -289.45) mm, rotated rx 81.04 ry 30.21 rz 20.91 deg; joints [-5.217, -0.415, 59.533, 103.38, 106.04, 56.915, -153.967]
  MoveL 7377 to (-57.99, 28.74, -289.43) mm, rotated rx 81.04 ry 30.21 rz 20.91 deg; joints [-5.222, -0.429, 59.519, 103.384, 106.036, 56.943, -153.967]
  MoveL 7378 to (-57.96, 28.44, -289.33) mm, rotated rx 81.04 ry 30.21 rz 20.91 deg; joints [-5.222, -0.441, 59.521, 103.387, 106.033, 56.954, -153.967]
  MoveL 7379 to (-58.01, 28.47, -289.13) mm, rotated rx 81.04 ry 30.21 rz 20.91 deg; joints [-5.218, -0.455, 59.548, 103.386, 106.034, 56.94, -153.967]
  MoveL 7380 to (-58.15, 28.88, -288.82) mm, rotated rx 81.04 ry 30.21 rz 20.91 deg; joints [-5.211, -0.472, 59.606, 103.381, 106.04, 56.898, -153.967]
  MoveL 7381 to (-58.52, 28.98, -288.2) mm, rotated rx 81.04 ry 30.21 rz 20.91 deg; joints [-5.192, -0.511, 59.682, 103.386, 106.04, 56.858, -153.967]
  MoveL 7382 to (-58.58, 26.94, -288.19) mm, rotated rx 81.04 ry 30.21 rz 20.91 deg; joints [-5.189, -0.532, 59.578, 103.423, 106.009, 56.984, -153.967]
  MoveL 7383 to (-58.73, 24.8, -288.14) mm, rotated rx 81.04 ry 30.21 rz 20.91 deg; joints [-5.183, -0.556, 59.471, 103.465, 105.976, 57.116, -153.967]
  MoveL 7384 to (-58.94, 22.54, -288.01) mm, rotated rx 81.04 ry 30.21 rz 20.91 deg; joints [-5.174, -0.583, 59.363, 103.51, 105.939, 57.252, -153.967]
  MoveL 7385 to (-59.14, 20.31, -287.91) mm, rotated rx 81.04 ry 30.21 rz 20.91 deg; joints [-5.166, -0.609, 59.254, 103.554, 105.904, 57.387, -153.967]
  MoveL 7386 to (-59.34, 18.17, -287.74) mm, rotated rx 81.04 ry 30.21 rz 20.91 deg; joints [-5.156, -0.639, 59.159, 103.596, 105.87, 57.512, -153.967]
  MoveL 7387 to (-59.52, 16.23, -287.59) mm, rotated rx 81.04 ry 30.21 rz 20.91 deg; joints [-5.148, -0.665, 59.071, 103.634, 105.839, 57.626, -153.967]
  MoveL 7388 to (-59.7, 14.17, -287.54) mm, rotated rx 81.04 ry 30.21 rz 20.91 deg; joints [-5.141, -0.684, 58.962, 103.675, 105.805, 57.755, -153.967]
  MoveL 7389 to (-59.88, 12.02, -287.47) mm, rotated rx 81.04 ry 30.21 rz 20.91 deg; joints [-5.134, -0.705, 58.85, 103.718, 105.77, 57.888, -153.967]
  MoveL 7390 to (-60.09, 9.68, -287.32) mm, rotated rx 81.04 ry 30.21 rz 20.91 deg; joints [-5.125, -0.734, 58.739, 103.764, 105.732, 58.028, -153.967]
  MoveL 7391 to (-60.25, 7.81, -287.2) mm, rotated rx 81.04 ry 30.21 rz 20.91 deg; joints [-5.117, -0.756, 58.648, 103.8, 105.701, 58.141, -153.967]
  MoveL 7392 to (-60.45, 5.43, -286.99) mm, rotated rx 81.04 ry 30.21 rz 20.91 deg; joints [-5.108, -0.789, 58.542, 103.846, 105.663, 58.28, -153.967]
  MoveL 7393 to (-60.61, 3.56, -286.88) mm, rotated rx 81.04 ry 30.21 rz 20.91 deg; joints [-5.101, -0.811, 58.451, 103.882, 105.632, 58.393, -153.967]
  MoveL 7394 to (-60.78, 1.43, -286.71) mm, rotated rx 81.04 ry 30.21 rz 20.91 deg; joints [-5.093, -0.838, 58.351, 103.923, 105.598, 58.519, -153.967]
  MoveL 7395 to (-60.98, -0.95, -286.66) mm, rotated rx 81.04 ry 30.21 rz 20.91 deg; joints [-5.085, -0.857, 58.219, 103.97, 105.557, 58.67, -153.967]
  MoveL 7396 to (-61.13, -2.82, -286.55) mm, rotated rx 81.04 ry 30.21 rz 20.91 deg; joints [-5.078, -0.877, 58.126, 104.006, 105.526, 58.783, -153.967]
  MoveL 7397 to (-61.29, -4.95, -286.39) mm, rotated rx 81.04 ry 30.21 rz 20.91 deg; joints [-5.071, -0.903, 58.025, 104.047, 105.491, 58.91, -153.967]
  MoveL 7398 to (-61.49, -7.33, -286.34) mm, rotated rx 81.04 ry 30.21 rz 20.91 deg; joints [-5.063, -0.92, 57.891, 104.093, 105.451, 59.062, -153.967]
  MoveL 7399 to (-61.63, -9.2, -286.22) mm, rotated rx 81.04 ry 30.21 rz 20.91 deg; joints [-5.057, -0.94, 57.796, 104.129, 105.419, 59.176, -153.967]
  MoveL 7400 to (-61.8, -11.42, -286.12) mm, rotated rx 81.04 ry 30.21 rz 20.91 deg; joints [-5.049, -0.96, 57.679, 104.172, 105.382, 59.313, -153.967]
  MoveL 7401 to (-61.98, -13.64, -286.05) mm, rotated rx 81.04 ry 30.21 rz 20.91 deg; joints [-5.042, -0.977, 57.555, 104.215, 105.344, 59.454, -153.967]
  MoveL 7402 to (-62.09, -15.51, -285.87) mm, rotated rx 81.04 ry 30.21 rz 20.91 deg; joints [-5.036, -1.002, 57.47, 104.249, 105.313, 59.564, -153.967]
  MoveL 7403 to (-62.17, -17.25, -285.62) mm, rotated rx 81.04 ry 30.21 rz 20.91 deg; joints [-5.03, -1.034, 57.406, 104.279, 105.286, 59.659, -153.967]
  MoveL 7404 to (-62.21, -18.87, -285.27) mm, rotated rx 81.04 ry 30.21 rz 20.91 deg; joints [-5.024, -1.074, 57.364, 104.306, 105.263, 59.74, -153.967]
  MoveL 7405 to (-61.68, -17.46, -284.58) mm, rotated rx 81.04 ry 30.21 rz 20.91 deg; joints [-5.033, -1.14, 57.576, 104.259, 105.304, 59.595, -153.967]
  MoveL 7406 to (-61.73, -17.68, -284.57) mm, rotated rx 81.04 ry 30.21 rz 20.91 deg; joints [-5.032, -1.14, 57.561, 104.265, 105.299, 59.61, -153.967]
  MoveL 7407 to (-61.85, -17.96, -284.56) mm, rotated rx 81.04 ry 30.21 rz 20.91 deg; joints [-5.028, -1.139, 57.541, 104.273, 105.292, 59.629, -153.967]
  MoveL 7408 to (-62.09, -18.35, -284.53) mm, rotated rx 81.04 ry 30.21 rz 20.91 deg; joints [-5.02, -1.137, 57.511, 104.287, 105.281, 59.656, -153.967]
  MoveL 7409 to (-62.39, -18.79, -284.49) mm, rotated rx 81.04 ry 30.21 rz 20.91 deg; joints [-5.01, -1.134, 57.475, 104.303, 105.268, 59.687, -153.967]
  MoveL 7410 to (-62.75, -19.29, -284.45) mm, rotated rx 81.04 ry 30.21 rz 20.91 deg; joints [-4.999, -1.13, 57.434, 104.322, 105.253, 59.723, -153.967]
  MoveL 7411 to (-64.39, -21.34, -284.45) mm, rotated rx 81.04 ry 30.21 rz 20.91 deg; joints [-4.948, -1.092, 57.228, 104.407, 105.184, 59.884, -153.967]
  MoveL 7412 to (-64.75, -21.82, -284.42) mm, rotated rx 81.04 ry 30.21 rz 20.91 deg; joints [-4.937, -1.087, 57.185, 104.426, 105.168, 59.92, -153.967]
  MoveL 7413 to (-65.16, -22.38, -284.36) mm, rotated rx 81.04 ry 30.21 rz 20.91 deg; joints [-4.924, -1.082, 57.14, 104.447, 105.151, 59.96, -153.967]
  MoveL 7414 to (-65.54, -22.88, -284.33) mm, rotated rx 81.04 ry 30.21 rz 20.91 deg; joints [-4.912, -1.077, 57.095, 104.466, 105.135, 59.997, -153.967]
  MoveL 7415 to (-65.86, -23.29, -284.33) mm, rotated rx 81.04 ry 30.21 rz 20.91 deg; joints [-4.901, -1.069, 57.054, 104.483, 105.121, 60.029, -153.967]
  MoveL 7416 to (-66.17, -23.67, -284.32) mm, rotated rx 81.04 ry 30.21 rz 20.91 deg; joints [-4.892, -1.062, 57.016, 104.499, 105.108, 60.059, -153.967]
  MoveL 7417 to (-66.5, -24.08, -284.32) mm, rotated rx 81.04 ry 30.21 rz 20.91 deg; joints [-4.882, -1.054, 56.974, 104.516, 105.094, 60.092, -153.967]
  MoveL 7418 to (-66.82, -24.48, -284.32) mm, rotated rx 81.04 ry 30.21 rz 20.91 deg; joints [-4.872, -1.047, 56.934, 104.532, 105.08, 60.123, -153.967]
  MoveL 7419 to (-67.11, -24.87, -284.29) mm, rotated rx 81.04 ry 30.21 rz 20.91 deg; joints [-4.863, -1.042, 56.899, 104.547, 105.068, 60.152, -153.967]
  MoveL 7420 to (-67.38, -25.24, -284.24) mm, rotated rx 81.04 ry 30.21 rz 20.91 deg; joints [-4.854, -1.04, 56.87, 104.561, 105.056, 60.178, -153.967]
  MoveL 7421 to (-67.69, -25.64, -284.22) mm, rotated rx 81.04 ry 30.21 rz 20.91 deg; joints [-4.844, -1.034, 56.833, 104.577, 105.043, 60.208, -153.967]
  MoveL 7422 to (-68.02, -26.05, -284.22) mm, rotated rx 81.04 ry 30.21 rz 20.91 deg; joints [-4.834, -1.027, 56.791, 104.594, 105.029, 60.24, -153.967]
  MoveL 7423 to (-68.67, -26.87, -284.22) mm, rotated rx 81.04 ry 30.21 rz 20.91 deg; joints [-4.814, -1.011, 56.707, 104.627, 105.001, 60.306, -153.967]
  Set speed (1000.0 mm/s)
  MoveL 7424 to (-86.38, -39.27, -284.22) mm, rotated rx 81.04 ry 30.21 rz 20.91 deg; joints [-4.279, -0.493, 54.955, 105.358, 104.386, 61.456, -153.967]
  Set speed (1000.0 mm/s)
  MoveL 7425 to (-86.38, -39.27, -284.22) mm, rotated rx 81.04 ry 30.21 rz 20.91 deg; joints [-4.279, -0.493, 54.955, 105.358, 104.386, 61.456, -153.967]
